Staubli VAL3: pp.pjx

--- pp.pjx ---
Parameters version=s7.1 stackSize=5000 millimeterUnit=true
Program file=Pick.pgx
Program file=Place.pgx
Program file=RobotMotion.pgx
Program file=start.pgx
Program file=stop.pgx
Data file=pp.dtx

--- pp.dtx ---
mdesc mNomSpeed
bool bBool1 = true
jointRx JHome
mdesc mSlow = {accel=25, vel=25, decel=25, tmax=25, rmax=25}
num nRep
pointRx pPointrx1[3]
  [0] = {fatherId=world[0]}
  [1] = {fatherId=world[0]}
  [2] = {fatherId=world[0]}
tool tTool1 = {fatherId=flange[0], ioLink=valve1}

--- Pick.pgx ---
program Pick(pointRx pPos)
begin
end
